VAR_GLOBAL
	gTime:	UDINT;
END_VAR

(* stored: Version 1.1.0.1, ProductVersion 3.1.4022.18
   GVL GVL: Id {ade82f02-21df-4b1e-b396-2c260dfaf950} *)
